(* IEC 61131-3 sources: ICSML/Codesys_V3/Function Blocks/Tanh_L.pou, 1 file *)

(* ---- Tanh_L.pou ---- *)
(*#-#-#-#-#-#-#-#-#-#---Declaration---#-#-#-#-#-#-#-#-#-#-#-#-#*)

(*
	Hyperbolic Tangent (Tanh) Activation Layer
*)
FUNCTION_BLOCK PUBLIC Tanh_L IMPLEMENTS Activation
VAR
	// Input and Output dataMem variables
	input_i: dataMem;
	output_i: dataMem;
END_VAR
(*#-#-#-#-#-#-#-#-#-#---Implementation---#-#-#-#-#-#-#-#-#-#-#-#-#*)
